Staubli VAL3: EDITSTR.pgx

public program editStr(string& x_sItem, string& x_sItemValue, num x_nSelect)
  local string l_sEmpty
  local num l_nKey
  local num l_nPos
begin
  //
  do
    call clear(0,13)
    call findPos(x_sItem,":",l_nPos)
    gotoxy(nTopX+1,nTopY+x_nSelect+1)
    setTextMode(0)
    put(x_sItem)
    call strlength(l_sEmpty,nBottomX-l_nPos+1)
    call type(nTopX+l_nPos+2,nTopY+x_nSelect+1,l_sEmpty)
    gotoxy(nTopX+l_nPos+2,nTopY+x_nSelect+1)
    l_nKey=get(x_sItemValue)
    call strfill(x_sItem,l_nPos+1,x_sItem)
    x_sItem=x_sItem+x_sItemValue
    call strlength(x_sItem,nBottomX+1)
    gotoxy(nTopX+1,nTopY+x_nSelect+1)
    setTextMode(1)
    call type(nTopX+1,nTopY+x_nSelect+1,x_sItem)
    setTextMode(0)
    delay(0)
  until l_nKey==270 or l_nKey==255
end
